(* PLC project cam_1dir_2speed, Dassault Systèmes ControlBuild 2024x *)
(* stored: creationDateTime 2023-10-03T11:13:20-01:00 *)

(* This module simulates the behaviour of a cam with 1 direction and 2 speeds (ovoid). *)
FUNCTION_BLOCK equipment_library.cam_1dir_2speed
  VAR_INPUT
    highSpeed : BOOL := false;
    lowSpeed : BOOL := false;
  END_VAR
  VAR_OUTPUT
    positionTranslat : REAL := 0.0;
    percentTranslat : REAL := 0.0;
    incrementTranslat : REAL := 0.0;
  END_VAR
  VAR_OUTPUT
    angleRotationDeg : REAL := 0.0;
    angleRotationRad : REAL := 0.0;
  END_VAR
  VAR
    firstCycle : BOOL := false;
    incrementRotation : REAL := 0.0;
    memoHs : BOOL := false;
    memoLs : BOOL := false;
    oldPosition : REAL := 0.0;
  END_VAR
  VAR CONSTANT
    maxTranslat : REAL := 1000.0;
    highSpeedVal : REAL := 2.0;
    initTranslat : REAL := 0.0;
    minTranslat : REAL := 0.0;
    lowSpeedVal : REAL := 1.0;
  END_VAR
  VAR
    d_locking : BOOL := false;
    v_d_locking : BOOL := false;
  END_VAR


ACTION C_source_code:
/* ----------------------------------------------------------------	*/
/* Type : Model of Operative Behaviour					*/
/* Category :  Actuators							*/
/* Author : Dassault Systemes						*/
/* Update date : June 2018							*/
/* ----------------------------------------------------------------	*/
/* This module simulate the behaviour of a cam with 1 direction and	*/
/* 2 speeds.									*/
/* The position of the cam goes from minTranslat to maxTranslat with	*/
/* 2 rotation speeds highSpeedVal et lowSpeedVal.			*/
/*										*/
/* nota : the starting position is forced by initTranslat.		*/
/* ----------------------------------------------------------------	*/

/* Declaration of variables which don't need to be visualized during simulation */
float pi=3.1415926;



/* ----------------------------------------------------------------	*/
/* Initialization of the position of the cam for the first step of	*/
/* simulation.								*/
/* ----------------------------------------------------------------	*/
if (! firstCycle) {
	if (initTranslat > maxTranslat) positionTranslat = maxTranslat;
	else
		if (initTranslat < minTranslat) positionTranslat = minTranslat;
		else positionTranslat = initTranslat;

	firstCycle = 1;
	if ((maxTranslat - minTranslat) != 0.0)
		angleRotationRad = acos(1 - ((positionTranslat - minTranslat)/(maxTranslat - minTranslat)*2.0));
}

/* ----------------------------------------------------------------	*/
/* Manage priorities of inputs' switching					*/
/* ----------------------------------------------------------------	*/
if (highSpeed && !memoLs) memoHs = 1;
if (!highSpeed) memoHs = 0;
if (!memoHs && lowSpeed) memoLs= 1;
if (!lowSpeed) memoLs = 0;


/* ----------------------------------------------------------------	*/
/* Rotation and translation (height of cam)				*/
/* ----------------------------------------------------------------	*/
if ((!d_locking) && (memoHs || memoLs)) {

	/* compute the increment of rotation according to the clock of simulation	*/
	if (memoHs) incrementRotation = highSpeedVal * (CLOCK_PERIOD/1000000);
	if (memoLs) incrementRotation = lowSpeedVal * (CLOCK_PERIOD/1000000);

	/* compute the angle of rotation (radian)	*/
	angleRotationRad = angleRotationRad + incrementRotation;
	if (angleRotationRad >= (2*pi)) {angleRotationRad -= 2*pi;}
	
	/* compute the position of translation	*/
	positionTranslat=(1 - cos(angleRotationRad))*(maxTranslat-minTranslat)/2.0 + minTranslat;
}

/* ----------------------------------------------------------------	*/
/* Compute the pecentage of height between the current position	*/
/* and the lowest and highest points of the cam				*/
/* ----------------------------------------------------------------	*/
percentTranslat = (100/(maxTranslat - minTranslat)) * (positionTranslat - minTranslat)  ;
		

/* ----------------------------------------------------------------	*/
/* Conversion of the rotation angle from radian to degree		*/
/* ----------------------------------------------------------------	*/
angleRotationDeg = (angleRotationRad*180)/pi;

/* ----------------------------------------------------------------	*/
/* Increment of translation							*/
/* ----------------------------------------------------------------	*/
incrementTranslat = positionTranslat - oldPosition;
oldPosition = positionTranslat;
END_ACTION

ACTION C_header:
#include <math.h>
END_ACTION
END_FUNCTION_BLOCK
